// Block: A0302_Spintore_PERS

DATA_BLOCK A0302_Spintore_PERS
VERSION : 0.1
   NON_RETAIN
   VAR
      Par : Struct
         Sens : Analogic_SensorManagement_Par;
      END_STRUCT;
      Data : Struct
         Sens : Analogic_SensorManagement_Data;
         HMI : HMI_Preset;
         Ax_Pos : A0301_Mach_Ax_Pos_Data;
      END_STRUCT;
      Par_Mach : A0301_Mach_Sens_Par;
      Par_Ax_Manu : Positioning_EPOS_Machine_Par;
      Pers_Data : Struct
         EncoderAbsolute_Preset_OK : Bool;
         Persistent_ActualPosition : LReal;
      END_STRUCT;
      Par_Ax_Auto : A0301_Mach_Speed_Par;
   END_VAR

BEGIN
   // No initialization required
END_DATA_BLOCK
